(* CODESYS project MNG_SimIO_Upd.export

Project tree, tasks and I/O mapping:
  MNG_SimIO/
    function block MNG_SIMIO_UPDATER [ST]
  data type MNG_APPLICATION_INPUTS_32BIT
  data type MNG_APPLICATION_OUTPUTS_32BIT
*)

// MNG_APPLICATION_INPUTS_32BIT
TYPE MNG_APPLICATION_INPUTS_32BIT :
STRUCT
    NumSignals                    : INT     := 14        ;
EndoflGreifarm01_ACT_SPD: REAL    := 0.0; (* aging_STEP_EndoflHubgeruest_EndoflGreifarm?KinSpeed *)

EndoflGreifarm01_DLT_POS: REAL    := 0.0; (* aging_STEP_EndoflHubgeruest_EndoflGreifarm?KinDelta *)

EndoflGreifarm01_AXIS: REAL    := 0.0; (* kaging_STEP_EndoflHubgeruest_EndoflGreifarm?KinAxis *)

EndoflHubgeruest01_AXIS: REAL    := 0.0; (* End_of_Line_Packaging_STEP_EndoflHubgeruest?KinAxis *)

EndoflHubgeruest01_DLT_POS: REAL    := 0.0; (* nd_of_Line_Packaging_STEP_EndoflHubgeruest?KinDelta *)

EndoflHubgeruest01_ACT_SPD: REAL    := 0.0; (* nd_of_Line_Packaging_STEP_EndoflHubgeruest?KinSpeed *)

EndoflGreifarm_RCHD: BOOL    := 0; (* ing_STEP_EndoflHubgeruest_EndoflGreifarm?KinReached *)

EndoflHubgeruest_RCHD: BOOL    := 0; (* _of_Line_Packaging_STEP_EndoflHubgeruest?KinReached *)

Sauger_VACUUM: BOOL    := 0; (* _STEP_EndoflHubgeruest_EndoflGreifarm_Sauger?Vacuum *)

EndoflSchieber_LBK: BOOL    := 0; (* ndoflGreifarm_Schieber_Hub_EndoflSchieber?KinAtBack *)

Virtueller_Greifer_VACUUM: BOOL    := 0; (* doflGreifarm_EndoflPlatte_Virtueller_Greifer?Vacuum *)

EndoflEnd_of_Line_Packaging_STEP_Status_in: UINT    := 0; (* _EndoflEnd_of_Line_Packaging_STEP?Status_in *)

EndoflEnd_of_Line_Packaging_STEP_Ausschieben_out: BOOL    := 0; (* _EndoflEnd_of_Line_Packaging_STEP?Ausschieben_out *)

EndoflLaufwagen_Hubausschiebpos: REAL    := 0.0; (* ng_STEP_Laufwagen_1_EndoflLaufwagen?Hubausschiebpos *)

END_STRUCT
END_TYPE

// MNG_APPLICATION_OUTPUTS_32BIT
TYPE MNG_APPLICATION_OUTPUTS_32BIT :
STRUCT
    NumSignals                    : INT     := 15        ;
EndoflGreifarm_TGT_POS: REAL    := 0.0; (* ging_STEP_EndoflHubgeruest_EndoflGreifarm?KinTarget *)

EndoflHubgeruest_TGT_POS: REAL    := 0.0; (* d_of_Line_Packaging_STEP_EndoflHubgeruest?KinTarget *)

Sauger_GRIP: BOOL    := 0; (* STEP_EndoflHubgeruest_EndoflGreifarm_Sauger?Gripper *)

Gleitschiene_Links_FWD: BOOL    := 0; (* eruest_EndoflGreifarm_Gleitschiene_Links?KinForward *)

Gleitschiene_Rechts_FWD: BOOL    := 0; (* ruest_EndoflGreifarm_Gleitschiene_Rechts?KinForward *)

Gleitschiene_Rechts_BWD: BOOL    := 0; (* bgeruest_EndoflGreifarm_Gleitschiene_Rechts?KinBack *)

Gleitschiene_Links_BWD: BOOL    := 0; (* ubgeruest_EndoflGreifarm_Gleitschiene_Links?KinBack *)

Schieber_Hub_BWD: BOOL    := 0; (* ndoflHubgeruest_EndoflGreifarm_Schieber_Hub?KinBack *)

Schieber_Hub_FWD: BOOL    := 0; (* flHubgeruest_EndoflGreifarm_Schieber_Hub?KinForward *)

EndoflZwischenlage_TRIG: BOOL    := 0; (* d_of_Line_Packaging_STEP_EndoflZwischenlage?Trigger *)

EndoflSchieber_FWD: BOOL    := 0; (* doflGreifarm_Schieber_Hub_EndoflSchieber?KinForward *)

EndoflSchieber_BWD: BOOL    := 0; (* _EndoflGreifarm_Schieber_Hub_EndoflSchieber?KinBack *)

Sink_Deactivate: BOOL    := 0; (* ng_STEP_EndoflEuro_laengs_800x1200_Sink?Deactivate *)

Gripper_GRIP: BOOL    := 0; (* ng_STEP_EndoflEuro_laengs_800x1200_Gripper?Gripper *)

Virtueller_Greifer_GRIP: BOOL    := 0; (* oflGreifarm_EndoflPlatte_Virtueller_Greifer?Gripper *)

END_STRUCT
END_TYPE

// MNG_SimIO/MNG_SIMIO_UPDATER
FUNCTION_BLOCK MNG_SIMIO_UPDATER
(* This function block implements simple TCP/IP client protocol.              *)
(* The max. size of binary tx/rx data has to be <= PLCPRJ_BUFFER_SIZE         *)
VAR_INPUT
connect : BOOL := FALSE;
IPAddress : STRING := '192.168.8.175';
port : INT := 5006;
timeout : DINT := 3;		(* Timeout in seconds *)
Q : MNG_Application_Outputs_32Bit;    (* Tx user data *)
END_VAR
VAR_OUTPUT
I      : MNG_Application_Inputs_32Bit        ; (* Rx user data *)
Counter   : DINT := 0;
Connected : BOOL := FALSE;
END_VAR
VAR
state : INT := 0;
socket : RTS_IEC_HANDLE := -1(*SOCKET_INVALID*);
bOptNoDelay: BOOL := TRUE;
sa:SOCKADDRESS;
fdRead:SOCKET_FD_SET;
tvTimeout:SOCKET_TIMEVAL;
pdiReady:DINT := 0;
toServer         : MNG_RawDatagram;
fromServer       : MNG_RawDatagram;
expectedSize, recvSize : LINT := 0;
sendSize: UDINT := 0; 
sentSize : LINT := 0;

bInit: BOOL := FALSE;
DWordBuffer      : DWORD                                               ; (* convert DWORD data *)
DIntBuffer       : DINT                                                ; (* convert DINT data *)
Segment11_F: BOOL;
Error: DINT;
diSocket: BOOL;
result: RTS_IEC_RESULT; 
callback: CB.CB_CALLBACK;
callbackError: CB.ERROR; 
END_VAR
(* @END_DECLARATION := '0'                                                    *)

IF NOT bInit THEN
//         SysCallbackRegister(INDEXOF(CallbackReset), EVENT_BEFORE_RESET);
	callback.eEvent := CB.EVENT.BEFORE_RESET;
	callback.eClass := CB.EVENT_CLASS.ALL_CLASSES;
	callback.eSource := CB.EVENT_SOURCE.ALL_SOURCES;
	callback.pPOUFunc := ADR(CallbackReset); 
	
	CB.RegisterCallback(callback, ADR(callbackError));
        bInit := TRUE;
END_IF
CASE state OF
0:											(* Init *)
  	socket := -1(*SOCKET_INVALID*);
  	Connected := FALSE;
  	IF connect THEN
  	        state  := 10;
  	END_IF
10:											(* Create socket *)
        socket := SysSockCreate(SOCKET_AF_INET, SOCKET_STREAM, 0, ADR(result));
        (*IF socket <> 0(*= SOCKET_INVALID*) THEN
            state := 100;
        ELSE
            state := 20;
        END_IF*)
		state := 20;
20:											(* Setup and Connect *)
        (* SysSockSetOption(socket, SOCKET_SOL, SOCKET_SO_SNDBUF, ADR(diMaxDataSize), SIZEOF(diMaxDataSize));
        SysSockSetOption(socket, SOCKET_SOL, SOCKET_SO_RCVBUF, ADR(diMaxDataSize), SIZEOF(diMaxDataSize));
        lOptLinger.l_onoff:=0;
        lOptLinger.l_linger:=0;
        SysSockSetOption(diSocket,	SOCKET_SOL, SOCKET_SO_LINGER, ADR(lOptLinger), SIZEOF(lOptLinger)); *)
        bOptNoDelay:=TRUE;
        SysSockSetOption(socket,	SOCKET_IPPROTO_TCP, SOCKET_TCP_NODELAY, ADR(bOptNoDelay), SIZEOF(bOptNoDelay));
        sa.sin_family:=SOCKET_AF_INET;
        sa.sin_addr.ulAddr:=GetIPAddress(IPAddress);
        tvTimeout.tv_sec := timeout ;
        tvTimeout.tv_usec := 0;
        fdRead.fd_count := 1;
        fdRead.fd_array[0] := socket;
        IF sa.sin_addr.ulAddr = SOCKET_INADDR_NONE THEN
                state := 121;
        ELSE
                 sa.sin_port:=SysSockHtons(port);
                 IF SysSockConnect(socket, ADR(sa), SIZEOF(sa)) = 0  THEN
                        state := 30;
                 ELSE
                         Error := 10035(*SysSockGetLastErrorSync(socket)*);	
						(* Query reason why connect reported failure *)
                                         CASE  Error OF
                         10035: 			(* EWOULDBLOCK *)
                                 state := 30;
                         10056: 			 (* ALREADY_CONNECTED*)
                                 state := 30;
                         ELSE
                                 state := 60;
                         END_CASE
                END_IF
        END_IF
30:											(* Data exchange *)
                Connected := TRUE;
                fdRead.fd_array[0] := socket;
                IF (SysSockSelect(SOCKET_FD_SETSIZE, ADR(fdRead), 0, 0, ADR(tvTimeout), ADR(pdiReady)) = CmpErrors.Errors.ERR_OK) AND pdiReady > 0 THEN
                expectedSize := 16 + (I.NumSignals+1) * 4;
                recvSize := SysSockRecv(socket, ADR(fromServer), expectedSize, 0, ADR(result));
                IF result <> CmpErrors.Errors.ERR_OK OR expectedSize <= 0 THEN
                         state := 60;

                ELSIF expectedSize = recvSize THEN

                        (* correct header data *)
                        fromServer.Header.ByteCount   	 := SysSockNtohl(fromServer.Header.ByteCount);
                        Counter                        				:= SysSockNtohl(fromServer.Header.Counter);
                        fromServer.Header.SentTime  	   := SysSockNtohl(fromServer.Header.SentTime);
                        fromServer.Header.DatagramType := SysSockNtohl(fromServer.Header.DatagramType);

                        (* currently only use the data on a 32 Bit raw image *)
                        IF fromServer.Header.DatagramType = MNG_DatagramType.MNG_Raw32BitImage THEN
                                                        (* REAL EndoflGreifarm01_ACT_SPD *)
                                                        DWordBuffer := SysSockNtohl(fromServer.Payload[2]);
                                                        SysMemCpy(pDest := ADR(I.EndoflGreifarm01_ACT_SPD), pSrc := ADR(DWordBuffer), udiCount := 4);
                                                        (* REAL EndoflGreifarm01_DLT_POS *)
                                                        DWordBuffer := SysSockNtohl(fromServer.Payload[3]);
                                                        SysMemCpy(pDest := ADR(I.EndoflGreifarm01_DLT_POS), pSrc := ADR(DWordBuffer), udiCount := 4);
                                                        (* REAL EndoflGreifarm01_AXIS *)
                                                        DWordBuffer := SysSockNtohl(fromServer.Payload[4]);
                                                        SysMemCpy(pDest := ADR(I.EndoflGreifarm01_AXIS), pSrc := ADR(DWordBuffer), udiCount := 4);
                                                        (* REAL EndoflHubgeruest01_AXIS *)
                                                        DWordBuffer := SysSockNtohl(fromServer.Payload[5]);
                                                        SysMemCpy(pDest := ADR(I.EndoflHubgeruest01_AXIS), pSrc := ADR(DWordBuffer), udiCount := 4);
                                                        (* REAL EndoflHubgeruest01_DLT_POS *)
                                                        DWordBuffer := SysSockNtohl(fromServer.Payload[6]);
                                                        SysMemCpy(pDest := ADR(I.EndoflHubgeruest01_DLT_POS), pSrc := ADR(DWordBuffer), udiCount := 4);
                                                        (* REAL EndoflHubgeruest01_ACT_SPD *)
                                                        DWordBuffer := SysSockNtohl(fromServer.Payload[7]);
                                                        SysMemCpy(pDest := ADR(I.EndoflHubgeruest01_ACT_SPD), pSrc := ADR(DWordBuffer), udiCount := 4);
                                                        (* BOOL EndoflGreifarm_RCHD *)
                                                        I.EndoflGreifarm_RCHD := fromServer.Payload[8] <> 0;
                                                        (* BOOL EndoflHubgeruest_RCHD *)
                                                        I.EndoflHubgeruest_RCHD := fromServer.Payload[9] <> 0;
                                                        (* BOOL Sauger_VACUUM *)
                                                        I.Sauger_VACUUM := fromServer.Payload[10] <> 0;
                                                        (* BOOL EndoflSchieber_LBK *)
                                                        I.EndoflSchieber_LBK := fromServer.Payload[11] <> 0;
                                                        (* BOOL Virtueller_Greifer_VACUUM *)
                                                        I.Virtueller_Greifer_VACUUM := fromServer.Payload[12] <> 0;
                                                        (* UINT EndoflEnd_of_Line_Packaging_STEP_Status_in *)
                                                        DWordBuffer := SysSockNtohl(fromServer.Payload[13]);
                                                        I.EndoflEnd_of_Line_Packaging_STEP_Status_in := DWORD_TO_UINT(DWordBuffer);
                                                        (* BOOL EndoflEnd_of_Line_Packaging_STEP_Ausschieben_out *)
                                                        I.EndoflEnd_of_Line_Packaging_STEP_Ausschieben_out := fromServer.Payload[14] <> 0;
                                                        (* REAL EndoflLaufwagen_Hubausschiebpos *)
                                                        DWordBuffer := SysSockNtohl(fromServer.Payload[15]);
                                                        SysMemCpy(pDest := ADR(I.EndoflLaufwagen_Hubausschiebpos), pSrc := ADR(DWordBuffer), udiCount := 4);
                                        state :=  40;
                END_IF
                END_IF
                ELSE
                state := 60;
                END_IF
40:											(* Send data *)
        sendSize := 16 + (Q.NumSignals+1) * 4;
        (*IF (SysSockSelect(SOCKET_FD_SETSIZE, ADR(fdRead), 0, 0, ADR(tvTimeout), ADR(result)) > 0) THEN*)
          toServer.Header.ByteCount    := SysSockHtonl(sendSize-16);
          toServer.Header.DatagramType := SysSockHtonl(MNG_DatagramType.MNG_Raw32BitImage);
          toServer.Header.Counter      := SysSockHtonl(Counter);
          toServer.Payload[1] := SysSockHtonl(Q.NumSignals); (* number of signals *)
                                                        (* REAL EndoflGreifarm_TGT_POS *)
                        SysMemCpy(pDest := ADR(DWordBuffer), pSrc := ADR(Q.EndoflGreifarm_TGT_POS), udiCount := 4);
                        toServer.Payload[2] := SysSockHtonl(DWordBuffer);
                                                        (* REAL EndoflHubgeruest_TGT_POS *)
                        SysMemCpy(pDest := ADR(DWordBuffer), pSrc := ADR(Q.EndoflHubgeruest_TGT_POS), udiCount := 4);
                        toServer.Payload[3] := SysSockHtonl(DWordBuffer);
                                                        (* BOOL Sauger_GRIP *)
                        IF Q.Sauger_GRIP = TRUE THEN
                            toServer.Payload[4] := 16#FFFFFFFF;   (*BOOL *)
                        ELSE
                            toServer.Payload[4] := 0;
                        END_IF;
                                                        (* BOOL Gleitschiene_Links_FWD *)
                        IF Q.Gleitschiene_Links_FWD = TRUE THEN
                            toServer.Payload[5] := 16#FFFFFFFF;   (*BOOL *)
                        ELSE
                            toServer.Payload[5] := 0;
                        END_IF;
                                                        (* BOOL Gleitschiene_Rechts_FWD *)
                        IF Q.Gleitschiene_Rechts_FWD = TRUE THEN
                            toServer.Payload[6] := 16#FFFFFFFF;   (*BOOL *)
                        ELSE
                            toServer.Payload[6] := 0;
                        END_IF;
                                                        (* BOOL Gleitschiene_Rechts_BWD *)
                        IF Q.Gleitschiene_Rechts_BWD = TRUE THEN
                            toServer.Payload[7] := 16#FFFFFFFF;   (*BOOL *)
                        ELSE
                            toServer.Payload[7] := 0;
                        END_IF;
                                                        (* BOOL Gleitschiene_Links_BWD *)
                        IF Q.Gleitschiene_Links_BWD = TRUE THEN
                            toServer.Payload[8] := 16#FFFFFFFF;   (*BOOL *)
                        ELSE
                            toServer.Payload[8] := 0;
                        END_IF;
                                                        (* BOOL Schieber_Hub_BWD *)
                        IF Q.Schieber_Hub_BWD = TRUE THEN
                            toServer.Payload[9] := 16#FFFFFFFF;   (*BOOL *)
                        ELSE
                            toServer.Payload[9] := 0;
                        END_IF;
                                                        (* BOOL Schieber_Hub_FWD *)
                        IF Q.Schieber_Hub_FWD = TRUE THEN
                            toServer.Payload[10] := 16#FFFFFFFF;   (*BOOL *)
                        ELSE
                            toServer.Payload[10] := 0;
                        END_IF;
                                                        (* BOOL EndoflZwischenlage_TRIG *)
                        IF Q.EndoflZwischenlage_TRIG = TRUE THEN
                            toServer.Payload[11] := 16#FFFFFFFF;   (*BOOL *)
                        ELSE
                            toServer.Payload[11] := 0;
                        END_IF;
                                                        (* BOOL EndoflSchieber_FWD *)
                        IF Q.EndoflSchieber_FWD = TRUE THEN
                            toServer.Payload[12] := 16#FFFFFFFF;   (*BOOL *)
                        ELSE
                            toServer.Payload[12] := 0;
                        END_IF;
                                                        (* BOOL EndoflSchieber_BWD *)
                        IF Q.EndoflSchieber_BWD = TRUE THEN
                            toServer.Payload[13] := 16#FFFFFFFF;   (*BOOL *)
                        ELSE
                            toServer.Payload[13] := 0;
                        END_IF;
                                                        (* BOOL Sink_Deactivate *)
                        IF Q.Sink_Deactivate = TRUE THEN
                            toServer.Payload[14] := 16#FFFFFFFF;   (*BOOL *)
                        ELSE
                            toServer.Payload[14] := 0;
                        END_IF;
                                                        (* BOOL Gripper_GRIP *)
                        IF Q.Gripper_GRIP = TRUE THEN
                            toServer.Payload[15] := 16#FFFFFFFF;   (*BOOL *)
                        ELSE
                            toServer.Payload[15] := 0;
                        END_IF;
                                                        (* BOOL Virtueller_Greifer_GRIP *)
                        IF Q.Virtueller_Greifer_GRIP = TRUE THEN
                            toServer.Payload[16] := 16#FFFFFFFF;   (*BOOL *)
                        ELSE
                            toServer.Payload[16] := 0;
                        END_IF;
        (*    toServer.Header.SentTime := SysSockHtonl(clock.systemTime.wMilliseconds + clock.systemTime.wMinute * 60000); *)
            sentSize := SysSockSend(socket, ADR(toServer), sendSize, 0, ADR(result));
            IF sentSize < 0 THEN
               state := 60;
            ELSE
               state := 30;
            END_IF
        (*ELSE
                        state := 60;
        END_IF*)
60:											(* Disconnect *)
                IF socket = 0(*SOCKET_INVALID*) THEN
                                state := 0;
                ELSE
                                IF SysSockClose(socket) <> 0(*= FALSE*) THEN
                                          state := 161;
                                ELSE
                                                state := 70;
                                END_IF
          END_IF
70:											(* Delete socket *)
          IF socket = 0(*SOCKET_INVALID*) THEN
                                state := 0;
                ELSE
                    IF SysSockShutdown(socket, 0) <> 0(*= FALSE*) THEN
                                          state := 0;
                                ELSE
                                                state := 0;
                                END_IF
          END_IF
110:										(* Error Create socket failed *)
;
121:										(* Error IP number invalid *)
;
122:										(* Error connect failed *)
     state := 70;
131:										(* Error while receiving, received bytes < expected)*)
                 state := 60;
161: 										(* Error close failed *)
;
END_CASE
IF NOT connect AND state> 0 AND state < 60 THEN
                state := 60;
END_IF

END_FUNCTION_BLOCK
